{attribute 'qualified_only'}
VAR_GLOBAL
	nTest AT %Q* : INT;
END_VAR

(* stored: Version 1.1.0.1, ProductVersion 3.1.4024.12
   GVL Test: Id {2c8fcf78-61e0-4aae-8078-f987169ea392} *)
